{attribute addProperty BoxType "EPP9022-0060-0017"}
{attribute addProperty Id "EPM_Inputs_ChannelAT %I*ARRAY[0..3] OF EPM_Inputs_Channel_19E518F4160200WcStateAT %I*WcState_98A4DF7520.250InfoDataAT %I*InfoData_BC63D37F80100"}
{attribute addProperty CRC "2919404861"}
{attribute addProperty SizeInBites "242"}
{attribute addProperty SizeInBytes "30.25"}
TYPE EPP9022_9F4D52F1 :
STRUCT
	{attribute addProperty Name "EPM_Inputs_Channel"}
	EPM_Inputs_Channel : ARRAY[0..3] OF EPM_Inputs_Channel_19E518F4;
	{attribute addProperty Name "WcState"}
	WcState : WcState_98A4DF75;
	{attribute addProperty Name "InfoData"}
	InfoData : InfoData_BC63D37F;
END_STRUCT
END_TYPE

(* stored: Version 1.2.0.0, ProductVersion 3.1.4024.9
   DUT EPP9022_9F4D52F1: Id {db3e5b9f-ac85-4455-932b-65f896fde6d9} *)
